# EPICS autosave request: ip/ipApp/Db/MPC_settings.req
#FILE... MPC_settings.req
#USAGE... MPC.db fields autosave'd.
$(P)$(PUMP)SAUTOS
$(P)$(PUMP)DIS
$(P)$(PUMP)SSIZE
$(P)$(PUMP)ULCK
$(P)$(PUMP)SIZE.SCAN
$(P)$(PUMP)STAT.SCAN
